(* IEC 61131-3 sources: stc/pkg/testing/testdata, 9 files *)

(* ---- mock_mc_moveabsolute.st ---- *)
FUNCTION_BLOCK MC_MoveAbsolute
VAR_INPUT
    Execute : BOOL;
    Position : LREAL;
END_VAR
VAR_OUTPUT
    Done : BOOL;
    Error : BOOL;
END_VAR
    Done := Execute;
    Error := FALSE;
END_FUNCTION_BLOCK

(* ---- stub_mc_moveabsolute.st ---- *)
FUNCTION_BLOCK MC_MoveAbsolute
VAR_INPUT
    Execute : BOOL;
    Position : LREAL;
END_VAR
VAR_OUTPUT
    Done : BOOL;
    Error : BOOL;
END_VAR
END_FUNCTION_BLOCK

(* ---- autostub_test.st ---- *)
TEST_CASE 'Auto-stub returns zero values'
VAR
    mover : MC_MoveAbsolute;
END_VAR
    mover(Execute := TRUE, Position := 100.0);
    ASSERT_FALSE(mover.Done, 'Auto-stub Done should be FALSE (zero)');
    ASSERT_FALSE(mover.Error, 'Auto-stub Error should be FALSE (zero)');
END_TEST_CASE

(* ---- failing_test.st ---- *)
TEST_CASE 'Intentional failure'
VAR
    x : INT := 1;
    y : INT := 2;
END_VAR
    ASSERT_EQ(x, y);
END_TEST_CASE

(* ---- io_inject_test.st ---- *)
TEST_CASE 'SET_IO and GET_IO work'
VAR
    sensor : BOOL;
END_VAR
    SET_IO('I', 0, 3, TRUE);
    sensor := GET_IO('I', 0, 3);
    ASSERT_TRUE(sensor, 'Should read back TRUE from I0.3');

    SET_IO('Q', 2, 0, TRUE);
    ASSERT_TRUE(GET_IO('Q', 2, 0), 'Should read back TRUE from Q2.0');
END_TEST_CASE

(* ---- mock_fb_test.st ---- *)
TEST_CASE 'Mock FB returns expected value'
VAR
    mover : MC_MoveAbsolute;
END_VAR
    mover(Execute := TRUE, Position := 100.0);
    ASSERT_TRUE(mover.Done, 'Mock should set Done to TRUE');
END_TEST_CASE

(* ---- multi_assert_test.st ---- *)
TEST_CASE 'Multiple assertions collected'
VAR
    x : INT := 10;
END_VAR
    ASSERT_TRUE(x > 5);
    ASSERT_EQ(x, 99);
    ASSERT_TRUE(x < 100);
END_TEST_CASE

(* ---- passing_test.st ---- *)
TEST_CASE 'Addition works'
VAR
    x : INT := 5;
    y : INT := 10;
    result : INT;
END_VAR
    result := x + y;
    ASSERT_EQ(result, 15);
    ASSERT_TRUE(result > 0);
END_TEST_CASE

TEST_CASE 'Boolean logic'
VAR
    a : BOOL := TRUE;
    b : BOOL := FALSE;
END_VAR
    ASSERT_TRUE(a);
    ASSERT_FALSE(b);
    ASSERT_EQ(a OR b, TRUE);
END_TEST_CASE

(* ---- timer_test.st ---- *)
TEST_CASE 'TON timer fires after preset'
VAR
    timer : TON;
    done : BOOL;
END_VAR
    timer(IN := TRUE, PT := T#100ms);
    ASSERT_FALSE(timer.Q);

    ADVANCE_TIME(T#50ms);
    timer(IN := TRUE, PT := T#100ms);
    ASSERT_FALSE(timer.Q);

    ADVANCE_TIME(T#60ms);
    timer(IN := TRUE, PT := T#100ms);
    ASSERT_TRUE(timer.Q);
END_TEST_CASE
